{attribute 'qualified_only'}
{attribute 'strict'}
{attribute 'to_string'}
TYPE E_SEQ_GENERAL :
(
	READY,
	EXECUTE,
	RESET,
	BUSY,
	DONE,
	ERROR,
	TIME_OUT	
);
END_TYPE

(* stored: Version 1.1.0.1, ProductVersion 3.1.4024.12
   EnumerationTextList E_SEQ_GENERAL: Id {a932f0ef-7aab-4ba2-973b-2cd37bdca6fc} *)
